(* PLC project SafeLOGIC, BrAutomation SafeDESIGNER  5.24.1.0 *)
(* stored: companyURL http://www.br-automation.com, creationDateTime Fri Nov 28 15:23:05 2025 *)

PROGRAM ERV_Lou

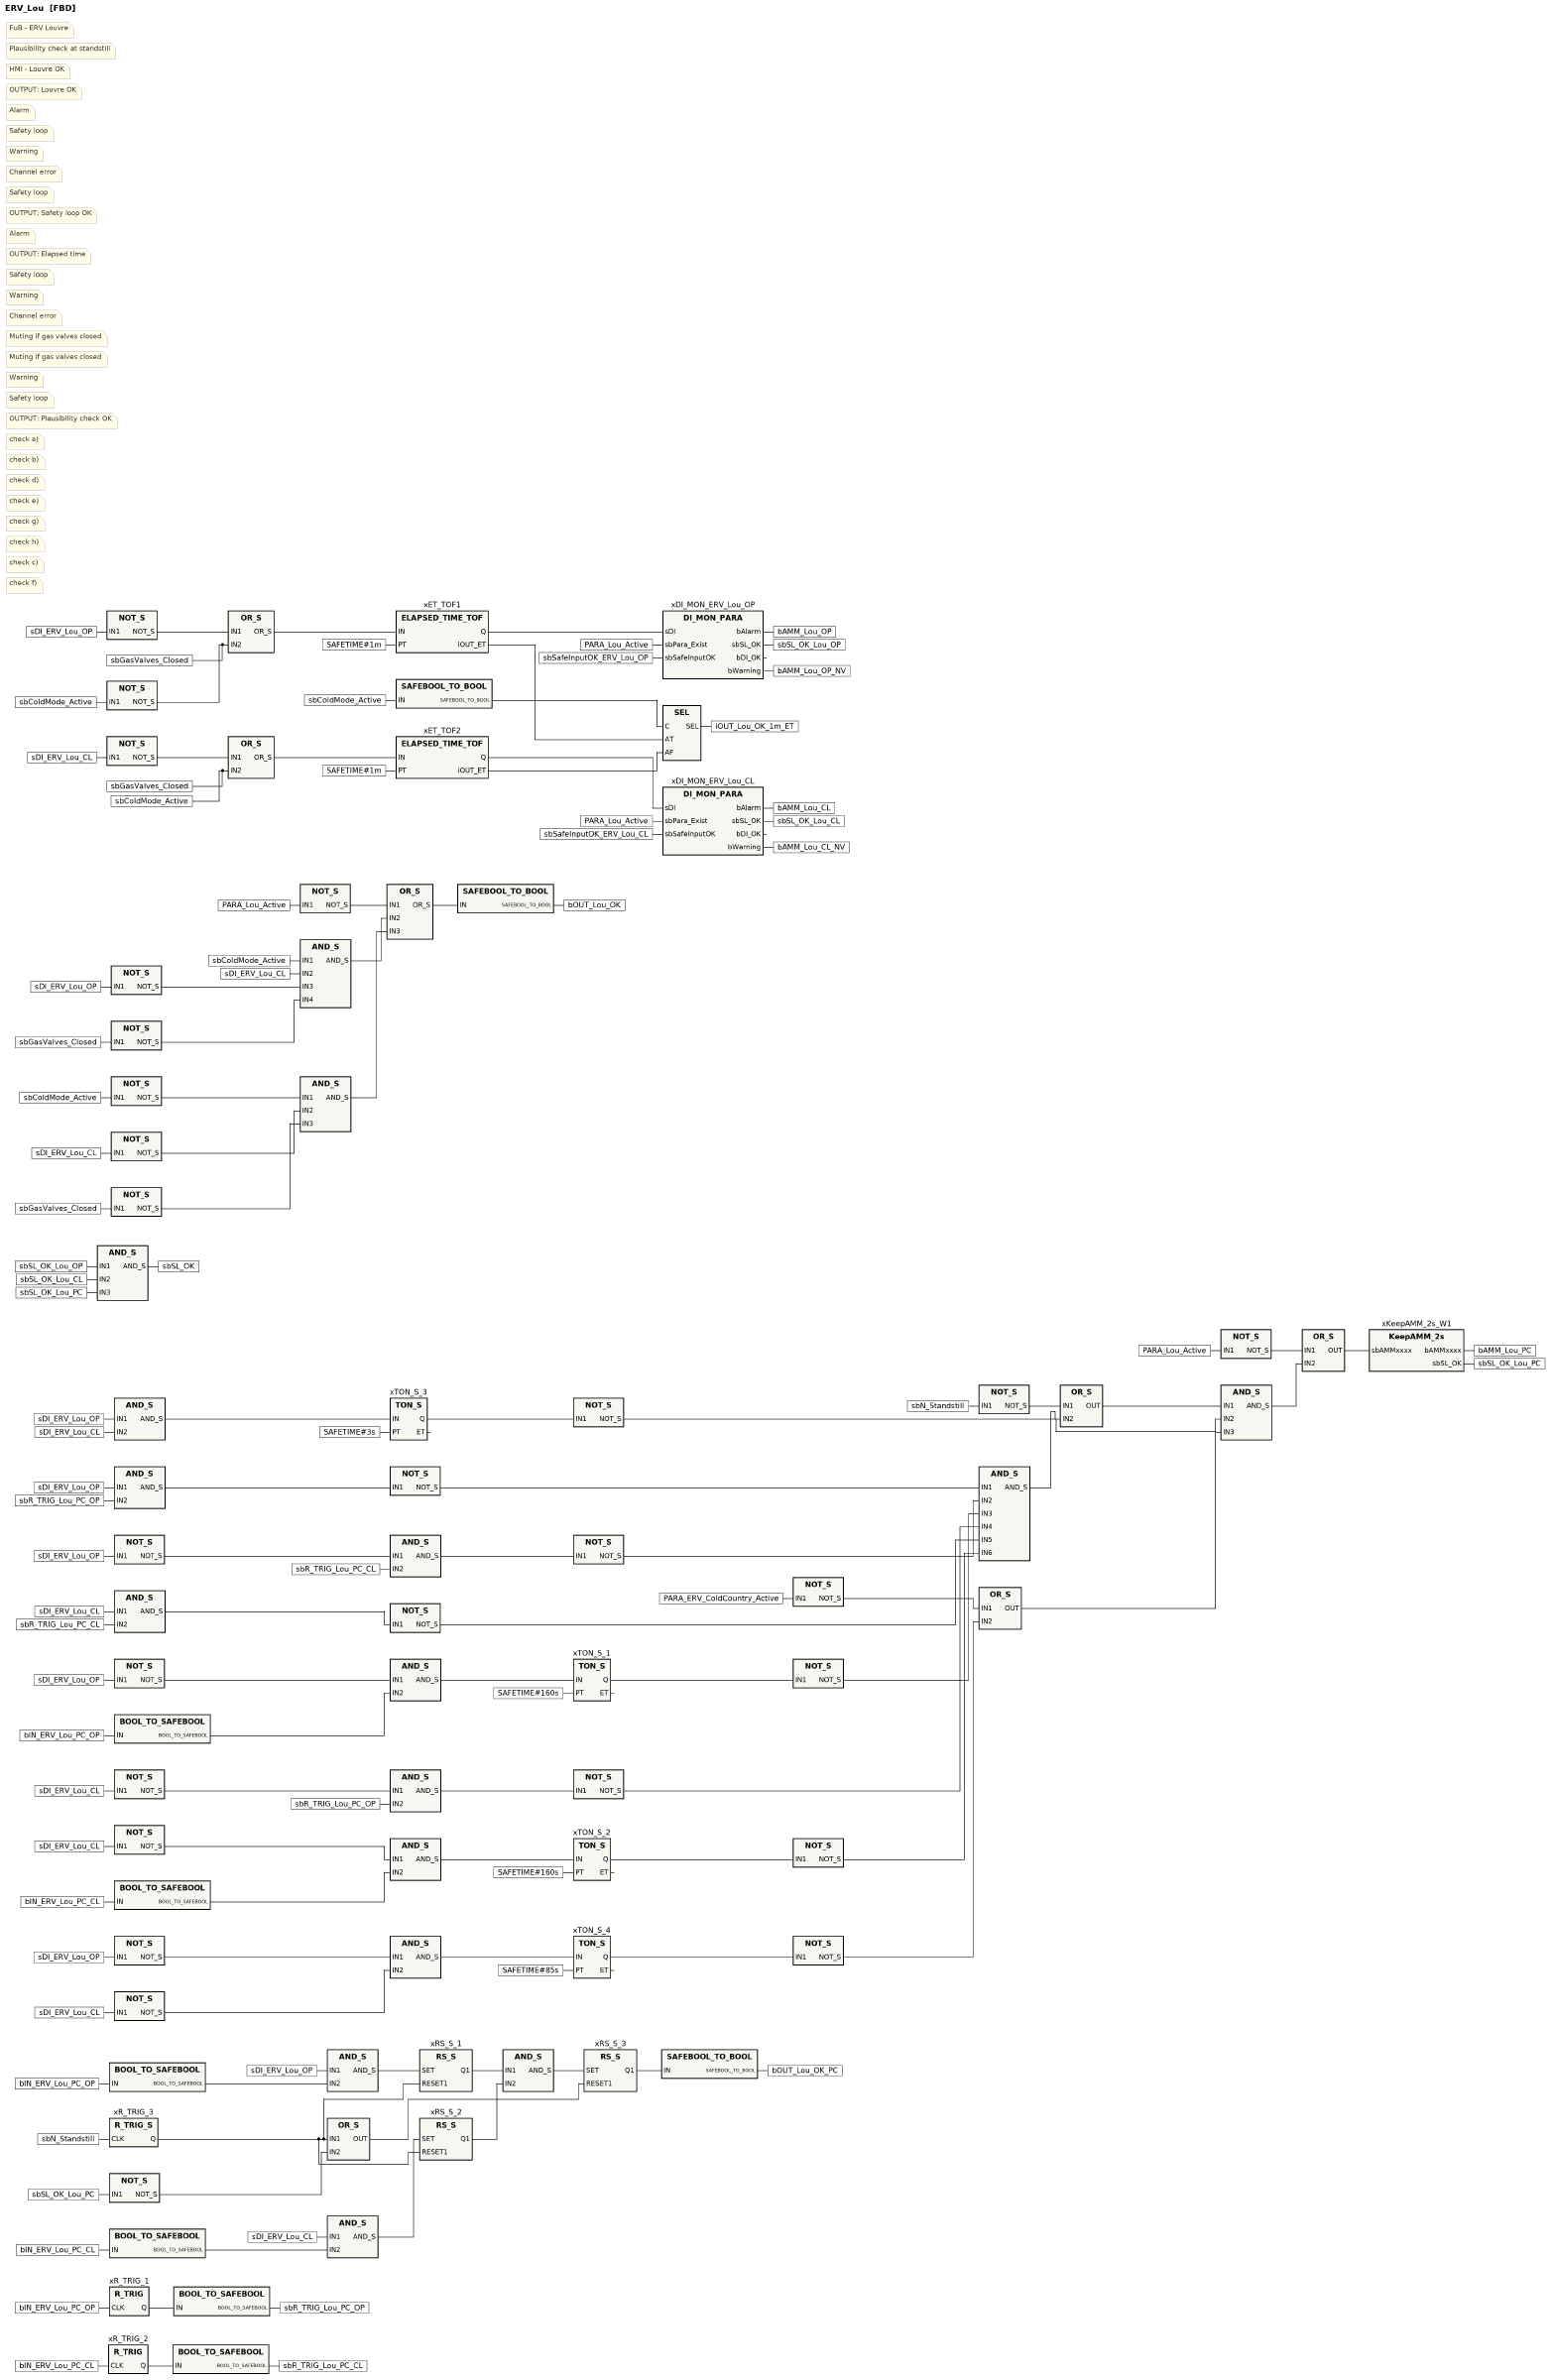
(* FBD diagram, written out as Structured Text *)
(* FuB - ERV Louvre *)
(* Alarm *)
(* Safety loop *)
xET_TOF1(IN := OR_S(NOT_S(sDI_ERV_Lou_OP), NOT_S(sbColdMode_Active), sbGasValves_Closed), PT := SAFETIME#1m);
xDI_MON_ERV_Lou_OP(sDI := xET_TOF1.Q, sbPara_Exist := PARA_Lou_Active, sbSafeInputOK := sbSafeInputOK_ERV_Lou_OP);
bAMM_Lou_OP := xDI_MON_ERV_Lou_OP.bAlarm;
(* Warning *)
(* Channel error *)
(* Muting if gas valves closed *)
bAMM_Lou_OP_NV := xDI_MON_ERV_Lou_OP.bWarning;
sbSL_OK_Lou_OP := xDI_MON_ERV_Lou_OP.sbSL_OK;
(* Alarm *)
(* Safety loop *)
xET_TOF2(IN := OR_S(NOT_S(sDI_ERV_Lou_CL), sbColdMode_Active, sbGasValves_Closed), PT := SAFETIME#1m);
xDI_MON_ERV_Lou_CL(sDI := xET_TOF2.Q, sbPara_Exist := PARA_Lou_Active, sbSafeInputOK := sbSafeInputOK_ERV_Lou_CL);
bAMM_Lou_CL := xDI_MON_ERV_Lou_CL.bAlarm;
(* Channel error *)
(* Muting if gas valves closed *)
(* Warning *)
bAMM_Lou_CL_NV := xDI_MON_ERV_Lou_CL.bWarning;
sbSL_OK_Lou_CL := xDI_MON_ERV_Lou_CL.sbSL_OK;
(* OUTPUT: Elapsed time *)
iOUT_Lou_OK_1m_ET := SEL(SAFEBOOL_TO_BOOL(sbColdMode_Active), xET_TOF1.iOUT_ET, xET_TOF2.iOUT_ET);
(* Plausibility check at standstill *)
xR_TRIG_1(CLK := bIN_ERV_Lou_PC_OP);
sbR_TRIG_Lou_PC_OP := BOOL_TO_SAFEBOOL(xR_TRIG_1.Q);
xR_TRIG_2(CLK := bIN_ERV_Lou_PC_CL);
sbR_TRIG_Lou_PC_CL := BOOL_TO_SAFEBOOL(xR_TRIG_2.Q);
(* Warning *)
(* Safety loop *)
xTON_S_1(IN := AND_S(NOT_S(sDI_ERV_Lou_OP), BOOL_TO_SAFEBOOL(bIN_ERV_Lou_PC_OP)), PT := SAFETIME#160s);
xTON_S_2(IN := AND_S(NOT_S(sDI_ERV_Lou_CL), BOOL_TO_SAFEBOOL(bIN_ERV_Lou_PC_CL)), PT := SAFETIME#160s);
xTON_S_3(IN := AND_S(sDI_ERV_Lou_OP, sDI_ERV_Lou_CL), PT := SAFETIME#3s);
xTON_S_4(IN := AND_S(NOT_S(sDI_ERV_Lou_OP), NOT_S(sDI_ERV_Lou_CL)), PT := SAFETIME#85s);
xKeepAMM_2s_W1(sbAMMxxxx := OR_S(NOT_S(PARA_Lou_Active), AND_S(OR_S(NOT_S(sbN_Standstill), AND_S(NOT_S(AND_S(sDI_ERV_Lou_OP, sbR_TRIG_Lou_PC_OP)), NOT_S(AND_S(NOT_S(sDI_ERV_Lou_OP), sbR_TRIG_Lou_PC_CL)), NOT_S(xTON_S_1.Q), NOT_S(AND_S(NOT_S(sDI_ERV_Lou_CL), sbR_TRIG_Lou_PC_OP)), NOT_S(AND_S(sDI_ERV_Lou_CL, sbR_TRIG_Lou_PC_CL)), NOT_S(xTON_S_2.Q))), NOT_S(xTON_S_3.Q), OR_S(NOT_S(PARA_ERV_ColdCountry_Active), NOT_S(xTON_S_4.Q)))));
bAMM_Lou_PC := xKeepAMM_2s_W1.bAMMxxxx;
sbSL_OK_Lou_PC := xKeepAMM_2s_W1.sbSL_OK;
(* check a) *)
(* check b) *)
(* check c) *)
(* check d) *)
(* check e) *)
(* check f) *)
(* check g) *)
(* check h) *)
(* OUTPUT: Plausibility check OK *)
xR_TRIG_3(CLK := sbN_Standstill);
xRS_S_1(SET := AND_S(sDI_ERV_Lou_OP, BOOL_TO_SAFEBOOL(bIN_ERV_Lou_PC_OP)), RESET1 := xR_TRIG_3.Q);
xRS_S_2(SET := AND_S(sDI_ERV_Lou_CL, BOOL_TO_SAFEBOOL(bIN_ERV_Lou_PC_CL)), RESET1 := xR_TRIG_3.Q);
xRS_S_3(SET := AND_S(xRS_S_1.Q1, xRS_S_2.Q1), RESET1 := OR_S(xR_TRIG_3.Q, NOT_S(sbSL_OK_Lou_PC)));
bOUT_Lou_OK_PC := SAFEBOOL_TO_BOOL(xRS_S_3.Q1);
(* HMI - Louvre OK *)
(* OUTPUT: Louvre OK *)
bOUT_Lou_OK := SAFEBOOL_TO_BOOL(OR_S(NOT_S(PARA_Lou_Active), AND_S(sbColdMode_Active, sDI_ERV_Lou_CL, NOT_S(sDI_ERV_Lou_OP), NOT_S(sbGasValves_Closed)), AND_S(NOT_S(sbColdMode_Active), NOT_S(sDI_ERV_Lou_CL), NOT_S(sbGasValves_Closed))));
(* Safety loop *)
(* OUTPUT: Safety loop OK *)
sbSL_OK := AND_S(sbSL_OK_Lou_OP, sbSL_OK_Lou_CL, sbSL_OK_Lou_PC);
END_PROGRAM
